FUNCTION_BLOCK PublishEventOpcUa (* Publish event using OPC UA *)
  (* Standard: 61499-2; Description: Copyright (c) 2019 fortiss GmbH This program and the accompanying materials are made available under the terms of the Eclipse Public License 2.0 which is available at https://www.eclipse.org/legal/epl-2.0/ SPDX-License-Identifier: EPL-2.0 *)
  (* Version 1.0, 2019-09-17, Cabral, fortiss GmbH *)
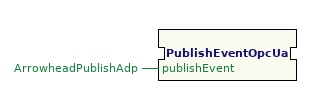
  SOCKETS
    publishEvent : ArrowheadPublishAdp; (* Publish Event adapter *)
  END_SOCKETS
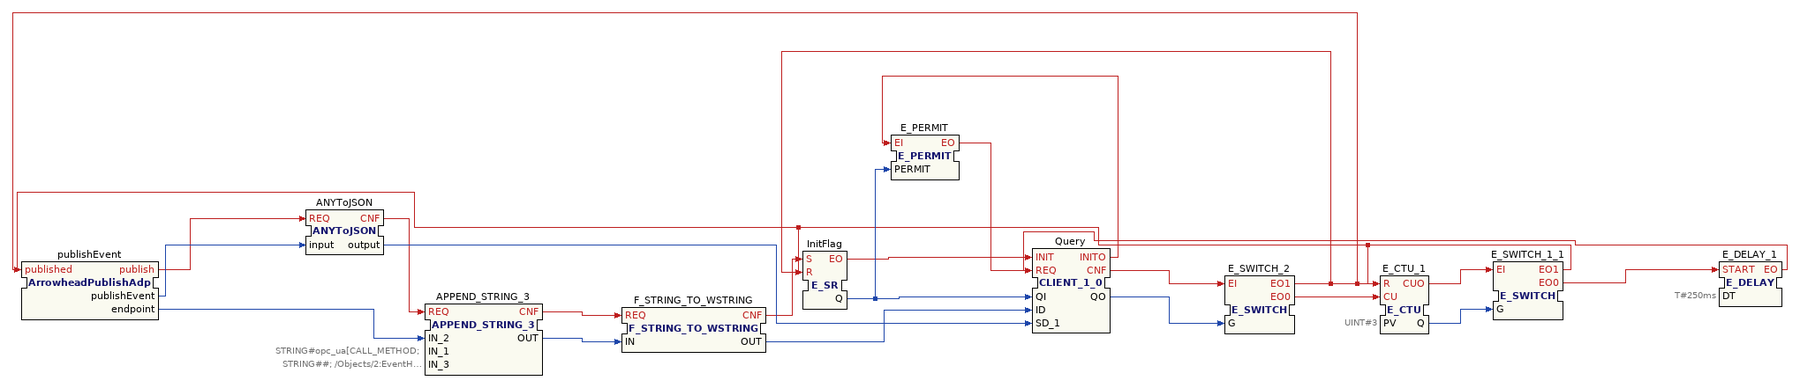
  FBS
    ANYToJSON : ANYToJSON;
    InitFlag : E_SR;
    APPEND_STRING_3 : APPEND_STRING_3(IN_1 := STRING#opc_ua[CALL_METHOD; , IN_3 := STRING##; /Objects/2:EventHandler/2:publish]);
    F_STRING_TO_WSTRING : F_STRING_TO_WSTRING;
    E_PERMIT : E_PERMIT;
    E_SWITCH_2 : E_SWITCH;
    E_SWITCH_1_1 : E_SWITCH;
    E_CTU_1 : E_CTU(PV := UINT#3);
    E_DELAY_1 : E_DELAY(DT := T#250ms);
    Query : CLIENT_1_0;
  END_FBS
  EVENT_CONNECTIONS
    APPEND_STRING_3.CNF TO F_STRING_TO_WSTRING.REQ;
    ANYToJSON.CNF TO APPEND_STRING_3.REQ;
    F_STRING_TO_WSTRING.CNF TO InitFlag.S;
    publishEvent.publish TO ANYToJSON.REQ;
    E_SWITCH_2.EO1 TO E_CTU_1.R;
    E_SWITCH_1_1.EO1 TO E_CTU_1.R;
    E_SWITCH_2.EO0 TO E_CTU_1.CU;
    E_CTU_1.CUO TO E_SWITCH_1_1.EI;
    E_SWITCH_1_1.EO0 TO E_DELAY_1.START;
    E_SWITCH_2.EO1 TO publishEvent.published;
    E_SWITCH_2.EO1 TO InitFlag.R;
    InitFlag.EO TO Query.INIT;
    E_PERMIT.EO TO Query.REQ;
    E_DELAY_1.EO TO Query.REQ;
    Query.INITO TO E_PERMIT.EI;
    Query.CNF TO E_SWITCH_2.EI;
    E_SWITCH_1_1.EO1 TO InitFlag.R;
    E_SWITCH_1_1.EO1 TO publishEvent.published;
  END_CONNECTIONS
  DATA_CONNECTIONS
    APPEND_STRING_3.OUT TO F_STRING_TO_WSTRING.IN;
    InitFlag.Q TO E_PERMIT.PERMIT;
    publishEvent.publishEvent TO ANYToJSON.input;
    publishEvent.endpoint TO APPEND_STRING_3.IN_2;
    E_CTU_1.Q TO E_SWITCH_1_1.G;
    InitFlag.Q TO Query.QI;
    F_STRING_TO_WSTRING.OUT TO Query.ID;
    ANYToJSON.output TO Query.SD_1;
    Query.QO TO E_SWITCH_2.G;
  END_CONNECTIONS
END_FUNCTION_BLOCK
